// TIA Portal V16 export
// export: Created 2022-02-04T14:40:23.5255935Z, ExportSetting WithDefaults, DisplayName Totally Integrated Automation Portal, DisplayVersion V16 Update 1, DisplayName TIA Portal Version Control Interface, DisplayVersion V16, DisplayName TIA Portal Openness, DisplayVersion V16, DisplayName SINAMICS Startdrive Advanced, DisplayVersion V16 Update 5, DisplayName SINAMICS Startdrive G130, G150, S120, S150, SINAMICS MV, S210, DisplayVersion V16 Update 5, DisplayName SINAMICS Startdrive G110M, G120, G120C, G120D, G120P, G115D, DisplayVersion V16 Update 5, DisplayName STEP 7 Professional, DisplayVersion V16, DisplayName STEP 7 Safety, DisplayVersion V16, DisplayName WinCC Advanced, DisplayVersion V16, DisplayName SIMATIC Visualization Architect, DisplayVersion V16
DATA_BLOCK "FB_Load_Zone_DB"   // DB30
VERSION : 0.1
// stored: AutoNumber true, InstanceOfName FB_Load_Zone, InstanceOfType FB
"FB_Load_Zone"
   // VAR RETAIN
   //    auto_mode_trigger : Bool;
   //    M213_mode : Bool;
   //    up_cmd_old : Bool;
   //    down_cmd_old : Bool;
   //    Lift_State : Int;
   //    Memento_Lift_State : Int;
   //    delayStart { S7_SetPoint := 'True'} : TON;
   //    wait_1 { S7_SetPoint := 'True'} : TOF;
   //    wait_2 { S7_SetPoint := 'True'} : TOF;
   //    wait_3 { S7_SetPoint := 'True'} : TOF;
   //    wait_213 { S7_SetPoint := 'True'} : TOF;
   // END_VAR
BEGIN
END_DATA_BLOCK
